FUNCTION_BLOCK EnOcean
VAR_INPUT
END_VAR
VAR_OUTPUT
END_VAR
VAR
	EnOceanRev: FB_KL6581;
	bReady: BOOL;
	bBusy: BOOL;
	bError: BOOL;
	iErrorID: INT;
END_VAR

//Initialize EnOcean gateway
EnOceanRev(
	bInit:= TRUE, 
	nIdx:= 1, 
	bReady=> bReady, 
	bBusy=> bBusy, 
	bError=> bError, 
	iErrorID=> iErrorID, 
	str_KL6581=> IO.str_KL6581, 
	stKL6581_in:= IO.stKL6581_In, 
	stKL6581_out:= IO.stKL6581_Out);

END_FUNCTION_BLOCK

(* stored: Version 1.1.0.1, ProductVersion 3.1.4022.16
   POU EnOcean: Id {ce5fd879-b97c-46fd-b6fd-2e37a62a2e0c}, SpecialFunc None *)
